{attribute 'qualified_only'}
{attribute 'strict'}
TYPE CAGroupStatus :
(
	mcGroupStateInvalid:=0, 
	mcGroupStateDisabled:=1,
	mcGroupStateStandby:=2, 
	mcGroupStateMoving:=3, 
	mcGroupStateStopping:=4, 
	mcGroupStateErrorStop:=5, 
	mcGroupStateHoming:=6, 
	mcGroupStateNotReady:=7, 
	mcGroupAllAxesStanding:=8,
    mcGroupConstantVelocity:=9,
    mcGroupAccelerating:=10,
    mcGroupDecelerating:=11,
    mcGroupInPosition:=12,
    mcGroupError:=13
);
END_TYPE

(* stored: Version 1.1.0.1
   DUT CAGroupStatus: Id {4279fe8e-03ff-4682-bd7f-b074d4f0a87e} *)
